Staubli VAL3: encodeStatus.pgx

public program encodeStatus()
begin
end
